// TIA Portal V17 export
// export: Created 2022-03-12T16:05:14.4802115Z, ExportSetting WithDefaults, DisplayName Totally Integrated Automation Portal, DisplayVersion V17, DisplayName TIA Portal Openness, DisplayVersion V17, DisplayName TIA Portal Version Control Interface, DisplayVersion V17, DisplayName STEP 7 Professional, DisplayVersion V17, DisplayName STEP 7 Safety, DisplayVersion V17, DisplayName WinCC Advanced / Unified PC, DisplayVersion V17
FUNCTION_BLOCK "UN_04_EventControl"   // FB31624, LAD
TITLE = UN_04_EventControl
{ S7_Optimized_Access := 'TRUE' }
AUTHOR : tech.team.motioncontrol@siemens.com
FAMILY : CPG
VERSION : 1.1
// Support: tech.team.motioncontrol@siemens.com
// stored: AutoNumber true, IsIECCheckEnabled false, IsRetainMemResEnabled false, MemoryReserve 100, SetENOAutomatically false, UDAEnableTagReadback false
   VAR
      instEventMgrAlarm { ExternalAccessible := 'False'; ExternalVisible := 'False'; ExternalWritable := 'False'; S7_SetPoint := 'True'} : "CPG_EventManager";   // instance FB - Event Manager - Alarms Events
      instEventMgrWarning { ExternalAccessible := 'False'; ExternalVisible := 'False'; ExternalWritable := 'False'; S7_SetPoint := 'True'} : "CPG_EventManager";   // instance FB - Event Manager - Warning Events
      instEventMgrStatus { ExternalAccessible := 'False'; ExternalVisible := 'False'; ExternalWritable := 'False'; S7_SetPoint := 'True'} : "CPG_EventManager";   // instance FB - Event Manager - Status Events
      instStatusAlarmsNotReset { ExternalAccessible := 'False'; ExternalVisible := 'False'; ExternalWritable := 'False'; S7_SetPoint := 'True'} : "CPG_Event";   // Status = Alarms Not Reset
      statEventMgr_Cmd_Reset { ExternalAccessible := 'False'; ExternalVisible := 'False'; ExternalWritable := 'False'} : Bool;   // Reset Cmd for event managers
      statEventMgr_Cmd_Clear1stFlt { ExternalAccessible := 'False'; ExternalVisible := 'False'; ExternalWritable := 'False'} : Bool;   // Clear 1st Fault Cmd for event managers
      statEventMgr_Clear1stFlt_OS { ExternalAccessible := 'False'; ExternalVisible := 'False'; ExternalWritable := 'False'} : Bool;   // Clear 1st Fault Cmd - One shot
   END_VAR
   VAR_TEMP   // added for the SCL form of the ladder/FBD networks
      _w1 : Bool;
      _w2 : Bool;
   END_VAR
BEGIN

REGION Network 2: ** STATE MODEL REPORTING STATUS ****
END_REGION

REGION Network 3: *** Call the PackML Module Initialize Logic ***
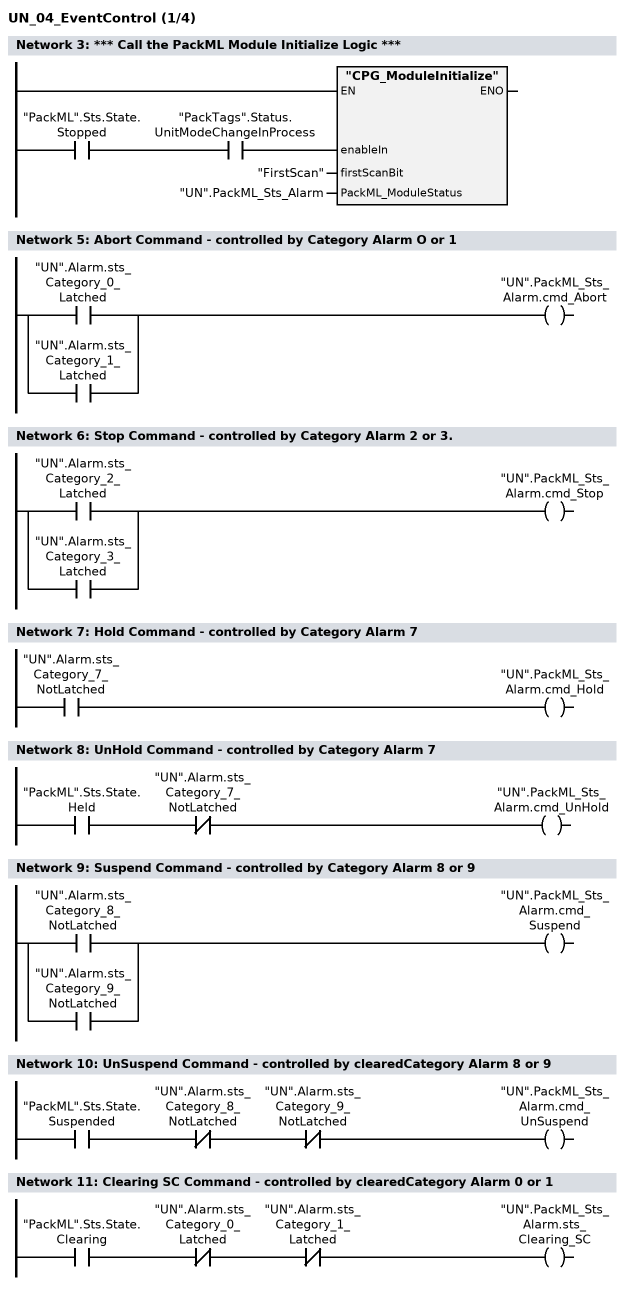
   RUNG wire#powerrail
      "CPG_ModuleInitialize"(enableIn := wire#w1, firstScanBit := "FirstScan", PackML_ModuleStatus := "UN".PackML_Sts_Alarm)
   END_RUNG
   RUNG wire#powerrail
      Contact( "PackML".Sts.State.Stopped )
      Contact( "PackTags".Status.UnitModeChangeInProcess )
   END_RUNG wire#w1
   // the same network as SCL:
   "CPG_ModuleInitialize"(enableIn := "PackML".Sts.State.Stopped AND "PackTags".Status.UnitModeChangeInProcess,
                          firstScanBit := "FirstScan",
                          PackML_ModuleStatus := "UN".PackML_Sts_Alarm);
END_REGION

REGION Network 4: Begin the LOGIC section.
END_REGION

REGION Network 5: Abort Command - controlled by Category Alarm O or 1
   RUNG wire#powerrail
      Contact( "UN".Alarm.sts_Category_0_Latched )
      wire#w1
      Coil( "UN".PackML_Sts_Alarm.cmd_Abort )
   END_RUNG
   RUNG wire#powerrail
      Contact( "UN".Alarm.sts_Category_1_Latched )
   END_RUNG wire#w1
   // the same network as SCL:
   "UN".PackML_Sts_Alarm.cmd_Abort := "UN".Alarm.sts_Category_0_Latched OR "UN".Alarm.sts_Category_1_Latched;
END_REGION

REGION Network 6: Stop Command - controlled by Category Alarm 2 or 3.
   RUNG wire#powerrail
      Contact( "UN".Alarm.sts_Category_2_Latched )
      wire#w1
      Coil( "UN".PackML_Sts_Alarm.cmd_Stop )
   END_RUNG
   RUNG wire#powerrail
      Contact( "UN".Alarm.sts_Category_3_Latched )
   END_RUNG wire#w1
   // the same network as SCL:
   "UN".PackML_Sts_Alarm.cmd_Stop := "UN".Alarm.sts_Category_2_Latched OR "UN".Alarm.sts_Category_3_Latched;
END_REGION

REGION Network 7: Hold Command - controlled by Category Alarm 7
   RUNG wire#powerrail
      Contact( "UN".Alarm.sts_Category_7_NotLatched )
      Coil( "UN".PackML_Sts_Alarm.cmd_Hold )
   END_RUNG
   // the same network as SCL:
   "UN".PackML_Sts_Alarm.cmd_Hold := "UN".Alarm.sts_Category_7_NotLatched;
END_REGION

REGION Network 8: UnHold Command - controlled by Category Alarm 7
   RUNG wire#powerrail
      Contact( "PackML".Sts.State.Held )
      I_Contact( "UN".Alarm.sts_Category_7_NotLatched )
      Coil( "UN".PackML_Sts_Alarm.cmd_UnHold )
   END_RUNG
   // the same network as SCL:
   "UN".PackML_Sts_Alarm.cmd_UnHold := "PackML".Sts.State.Held AND NOT "UN".Alarm.sts_Category_7_NotLatched;
END_REGION

REGION Network 9: Suspend Command - controlled by Category Alarm 8 or 9
   RUNG wire#powerrail
      Contact( "UN".Alarm.sts_Category_8_NotLatched )
      wire#w1
      Coil( "UN".PackML_Sts_Alarm.cmd_Suspend )
   END_RUNG
   RUNG wire#powerrail
      Contact( "UN".Alarm.sts_Category_9_NotLatched )
   END_RUNG wire#w1
   // the same network as SCL:
   "UN".PackML_Sts_Alarm.cmd_Suspend := "UN".Alarm.sts_Category_8_NotLatched OR "UN".Alarm.sts_Category_9_NotLatched;
END_REGION

REGION Network 10: UnSuspend Command - controlled by clearedCategory Alarm 8 or 9
   RUNG wire#powerrail
      Contact( "PackML".Sts.State.Suspended )
      I_Contact( "UN".Alarm.sts_Category_8_NotLatched )
      I_Contact( "UN".Alarm.sts_Category_9_NotLatched )
      Coil( "UN".PackML_Sts_Alarm.cmd_UnSuspend )
   END_RUNG
   // the same network as SCL:
   "UN".PackML_Sts_Alarm.cmd_UnSuspend := "PackML".Sts.State.Suspended AND NOT "UN".Alarm.sts_Category_8_NotLatched AND NOT "UN".Alarm.sts_Category_9_NotLatched;
END_REGION

REGION Network 11: Clearing SC Command - controlled by clearedCategory Alarm 0 or 1
   RUNG wire#powerrail
      Contact( "PackML".Sts.State.Clearing )
      I_Contact( "UN".Alarm.sts_Category_0_Latched )
      I_Contact( "UN".Alarm.sts_Category_1_Latched )
      Coil( "UN".PackML_Sts_Alarm.sts_Clearing_SC )
   END_RUNG
   // the same network as SCL:
   "UN".PackML_Sts_Alarm.sts_Clearing_SC := "PackML".Sts.State.Clearing AND NOT "UN".Alarm.sts_Category_0_Latched AND NOT "UN".Alarm.sts_Category_1_Latched;
END_REGION

REGION Network 12: Resetting S Command - controlled by clearedCategory Alarm 0-4
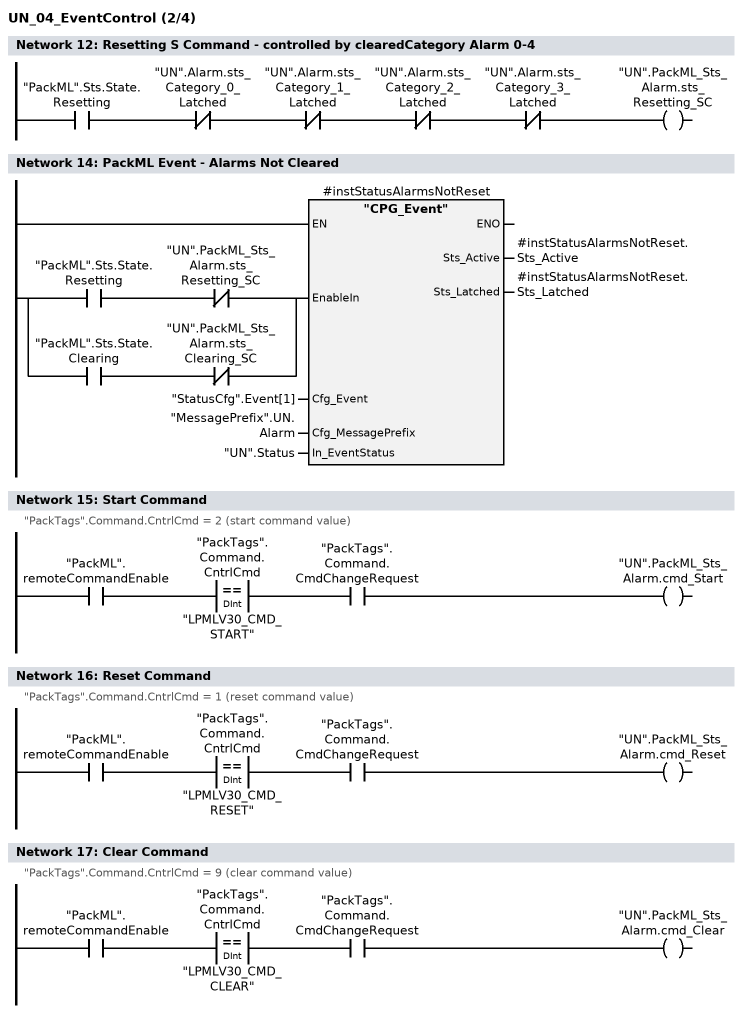
   RUNG wire#powerrail
      Contact( "PackML".Sts.State.Resetting )
      I_Contact( "UN".Alarm.sts_Category_0_Latched )
      I_Contact( "UN".Alarm.sts_Category_1_Latched )
      I_Contact( "UN".Alarm.sts_Category_2_Latched )
      I_Contact( "UN".Alarm.sts_Category_3_Latched )
      Coil( "UN".PackML_Sts_Alarm.sts_Resetting_SC )
   END_RUNG
   // the same network as SCL:
   "UN".PackML_Sts_Alarm.sts_Resetting_SC := "PackML".Sts.State.Resetting AND NOT "UN".Alarm.sts_Category_0_Latched AND NOT "UN".Alarm.sts_Category_1_Latched AND NOT "UN".Alarm.sts_Category_2_Latched AND NOT "UN".Alarm.sts_Category_3_Latched;
END_REGION

REGION Network 13: PackML Event -
END_REGION

REGION Network 14: PackML Event - Alarms Not Cleared
   RUNG wire#powerrail
      #instStatusAlarmsNotReset(EnableIn := wire#w1, Cfg_Event := "StatusCfg".Event[1], Cfg_MessagePrefix := "MessagePrefix".UN.Alarm, In_EventStatus := "UN".Status, Sts_Active => #instStatusAlarmsNotReset.Sts_Active, Sts_Latched => #instStatusAlarmsNotReset.Sts_Latched)
   END_RUNG
   RUNG wire#powerrail
      Contact( "PackML".Sts.State.Resetting )
      I_Contact( "UN".PackML_Sts_Alarm.sts_Resetting_SC )
   END_RUNG wire#w1
   RUNG wire#powerrail
      Contact( "PackML".Sts.State.Clearing )
      I_Contact( "UN".PackML_Sts_Alarm.sts_Clearing_SC )
   END_RUNG wire#w1
   // the same network as SCL:
   #instStatusAlarmsNotReset(EnableIn := ("PackML".Sts.State.Resetting AND NOT "UN".PackML_Sts_Alarm.sts_Resetting_SC) OR ("PackML".Sts.State.Clearing AND NOT "UN".PackML_Sts_Alarm.sts_Clearing_SC),   // "CPG_Event"
                           Cfg_Event := "StatusCfg".Event[1],
                           Cfg_MessagePrefix := "MessagePrefix".UN.Alarm,
                           In_EventStatus := "UN".Status,
                           Sts_Active => #instStatusAlarmsNotReset.Sts_Active,
                           Sts_Latched => #instStatusAlarmsNotReset.Sts_Latched);
END_REGION

REGION Network 15: Start Command
   // "PackTags".Command.CntrlCmd = 2 (start command value)
   RUNG wire#powerrail
      Contact( "PackML".remoteCommandEnable )
      { S7_Templates := "SrcType := DInt" } EQ_Contact(in1 := "PackTags".Command.CntrlCmd, in2 := "LPMLV30_CMD_START")
      Contact( "PackTags".Command.CmdChangeRequest )
      Coil( "UN".PackML_Sts_Alarm.cmd_Start )
   END_RUNG
   // the same network as SCL:
   "UN".PackML_Sts_Alarm.cmd_Start := "PackML".remoteCommandEnable AND ("PackTags".Command.CntrlCmd = "LPMLV30_CMD_START") AND "PackTags".Command.CmdChangeRequest;
END_REGION

REGION Network 16: Reset Command
   // "PackTags".Command.CntrlCmd = 1 (reset command value)
   RUNG wire#powerrail
      Contact( "PackML".remoteCommandEnable )
      { S7_Templates := "SrcType := DInt" } EQ_Contact(in1 := "PackTags".Command.CntrlCmd, in2 := "LPMLV30_CMD_RESET")
      Contact( "PackTags".Command.CmdChangeRequest )
      Coil( "UN".PackML_Sts_Alarm.cmd_Reset )
   END_RUNG
   // the same network as SCL:
   "UN".PackML_Sts_Alarm.cmd_Reset := "PackML".remoteCommandEnable AND ("PackTags".Command.CntrlCmd = "LPMLV30_CMD_RESET") AND "PackTags".Command.CmdChangeRequest;
END_REGION

REGION Network 17: Clear Command
   // "PackTags".Command.CntrlCmd = 9 (clear command value)
   RUNG wire#powerrail
      Contact( "PackML".remoteCommandEnable )
      { S7_Templates := "SrcType := DInt" } EQ_Contact(in1 := "PackTags".Command.CntrlCmd, in2 := "LPMLV30_CMD_CLEAR")
      Contact( "PackTags".Command.CmdChangeRequest )
      Coil( "UN".PackML_Sts_Alarm.cmd_Clear )
   END_RUNG
   // the same network as SCL:
   "UN".PackML_Sts_Alarm.cmd_Clear := "PackML".remoteCommandEnable AND ("PackTags".Command.CntrlCmd = "LPMLV30_CMD_CLEAR") AND "PackTags".Command.CmdChangeRequest;
END_REGION

REGION Network 18: *** EVENT CONTROL MANAGERS ***
END_REGION

REGION Network 19: Reset Command - for all event managers
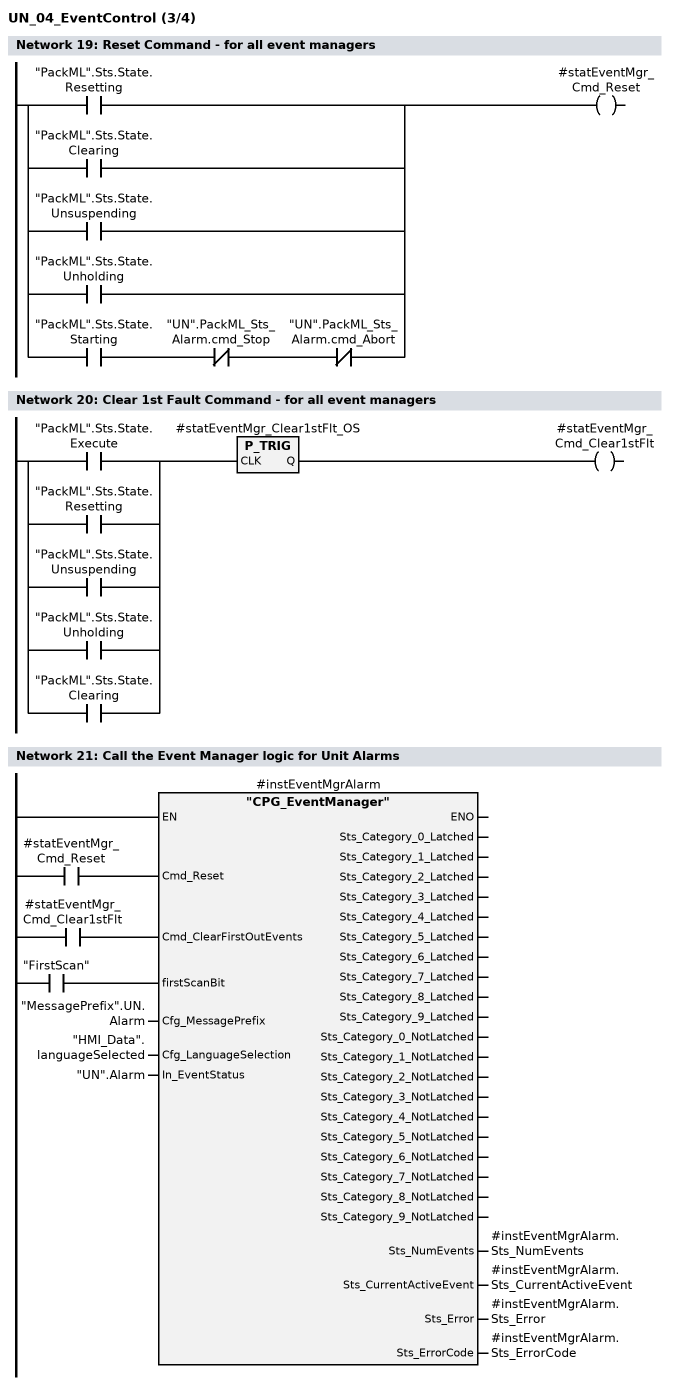
   RUNG wire#powerrail
      Contact( "PackML".Sts.State.Resetting )
      wire#w1
      Coil( #statEventMgr_Cmd_Reset )
   END_RUNG
   RUNG wire#powerrail
      Contact( "PackML".Sts.State.Clearing )
   END_RUNG wire#w1
   RUNG wire#powerrail
      Contact( "PackML".Sts.State.Unsuspending )
   END_RUNG wire#w1
   RUNG wire#powerrail
      Contact( "PackML".Sts.State.Unholding )
   END_RUNG wire#w1
   RUNG wire#powerrail
      Contact( "PackML".Sts.State.Starting )
      I_Contact( "UN".PackML_Sts_Alarm.cmd_Stop )
      I_Contact( "UN".PackML_Sts_Alarm.cmd_Abort )
   END_RUNG wire#w1
   // the same network as SCL:
   #statEventMgr_Cmd_Reset := "PackML".Sts.State.Resetting OR "PackML".Sts.State.Clearing OR "PackML".Sts.State.Unsuspending OR "PackML".Sts.State.Unholding OR ("PackML".Sts.State.Starting AND NOT "UN".PackML_Sts_Alarm.cmd_Stop AND NOT "UN".PackML_Sts_Alarm.cmd_Abort);
END_REGION

REGION Network 20: Clear 1st Fault Command - for all event managers
   RUNG wire#powerrail
      Contact( "PackML".Sts.State.Execute )
      wire#w1
      P_Trig( #statEventMgr_Clear1stFlt_OS )
      Coil( #statEventMgr_Cmd_Clear1stFlt )
   END_RUNG
   RUNG wire#powerrail
      Contact( "PackML".Sts.State.Resetting )
   END_RUNG wire#w1
   RUNG wire#powerrail
      Contact( "PackML".Sts.State.Unsuspending )
   END_RUNG wire#w1
   RUNG wire#powerrail
      Contact( "PackML".Sts.State.Unholding )
   END_RUNG wire#w1
   RUNG wire#powerrail
      Contact( "PackML".Sts.State.Clearing )
   END_RUNG wire#w1
   // the same network as SCL:
   #_w1 := "PackML".Sts.State.Execute OR "PackML".Sts.State.Resetting OR "PackML".Sts.State.Unsuspending OR "PackML".Sts.State.Unholding OR "PackML".Sts.State.Clearing;
   #_w2 := #_w1 AND NOT #statEventMgr_Clear1stFlt_OS;   // rising edge
   #statEventMgr_Clear1stFlt_OS := #_w1;
   #statEventMgr_Cmd_Clear1stFlt := #_w2;
END_REGION

REGION Network 21: Call the Event Manager logic for Unit Alarms
   RUNG wire#powerrail
      #instEventMgrAlarm(Cmd_Reset := wire#w1, Cmd_ClearFirstOutEvents := wire#w2, firstScanBit := wire#w3, Cfg_MessagePrefix := "MessagePrefix".UN.Alarm, Cfg_LanguageSelection := "HMI_Data".languageSelected, In_EventStatus := "UN".Alarm, Sts_Category_0_Latched =>, Sts_Category_1_Latched =>, Sts_Category_2_Latched =>, Sts_Category_3_Latched =>, Sts_Category_4_Latched =>, Sts_Category_5_Latched =>, Sts_Category_6_Latched =>, Sts_Category_7_Latched =>, Sts_Category_8_Latched =>, Sts_Category_9_Latched =>, Sts_Category_0_NotLatched =>, Sts_Category_1_NotLatched =>, Sts_Category_2_NotLatched =>, Sts_Category_3_NotLatched =>, Sts_Category_4_NotLatched =>, Sts_Category_5_NotLatched =>, Sts_Category_6_NotLatched =>, Sts_Category_7_NotLatched =>, Sts_Category_8_NotLatched =>, Sts_Category_9_NotLatched =>, Sts_NumEvents => #instEventMgrAlarm.Sts_NumEvents, Sts_CurrentActiveEvent => #instEventMgrAlarm.Sts_CurrentActiveEvent, Sts_Error => #instEventMgrAlarm.Sts_Error, Sts_ErrorCode => #instEventMgrAlarm.Sts_ErrorCode)
   END_RUNG
   RUNG wire#powerrail
      Contact( #statEventMgr_Cmd_Reset )
   END_RUNG wire#w1
   RUNG wire#powerrail
      Contact( #statEventMgr_Cmd_Clear1stFlt )
   END_RUNG wire#w2
   RUNG wire#powerrail
      Contact( "FirstScan" )
   END_RUNG wire#w3
   // the same network as SCL:
   #instEventMgrAlarm(Cmd_Reset := #statEventMgr_Cmd_Reset,   // "CPG_EventManager"
                      Cmd_ClearFirstOutEvents := #statEventMgr_Cmd_Clear1stFlt,
                      firstScanBit := "FirstScan",
                      Cfg_MessagePrefix := "MessagePrefix".UN.Alarm,
                      Cfg_LanguageSelection := "HMI_Data".languageSelected,
                      In_EventStatus := "UN".Alarm,
                      Sts_NumEvents => #instEventMgrAlarm.Sts_NumEvents,
                      Sts_CurrentActiveEvent => #instEventMgrAlarm.Sts_CurrentActiveEvent,
                      Sts_Error => #instEventMgrAlarm.Sts_Error,
                      Sts_ErrorCode => #instEventMgrAlarm.Sts_ErrorCode);
END_REGION

REGION Network 22: Call the Event Manager logic for Unit Warnings
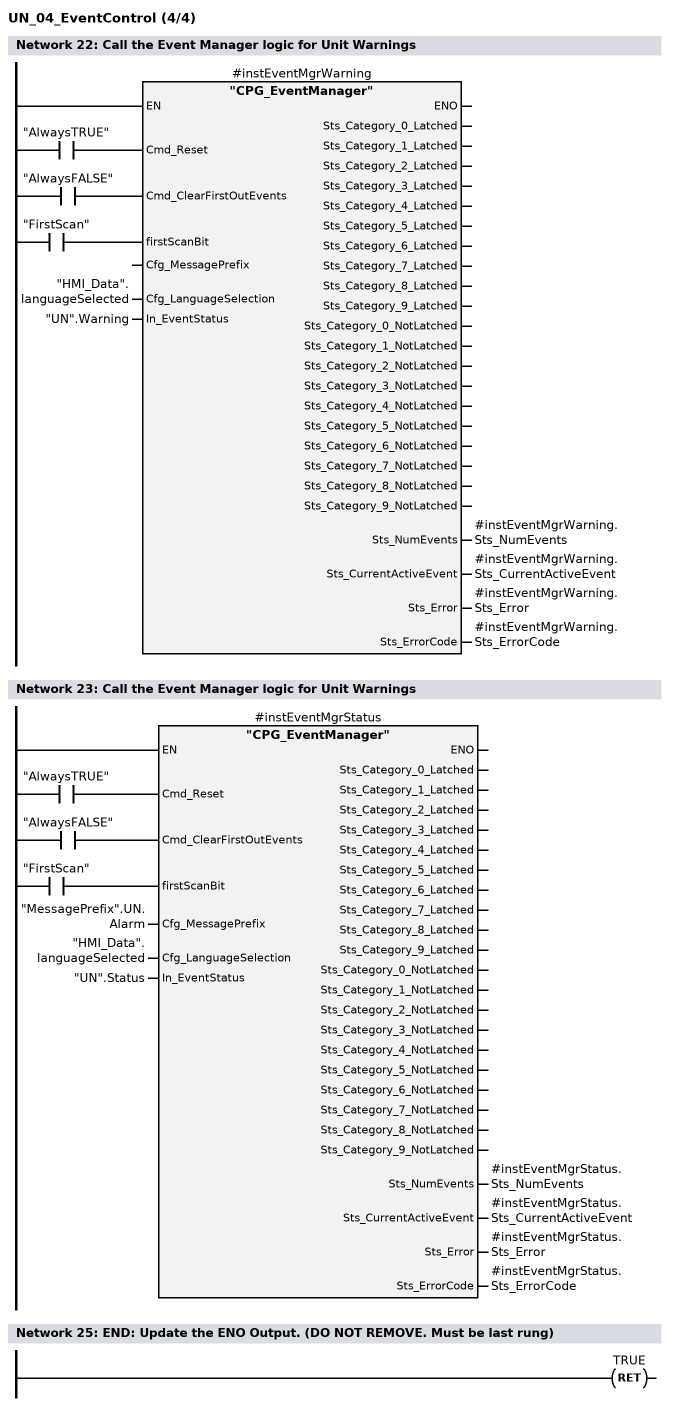
   RUNG wire#powerrail
      #instEventMgrWarning(Cmd_Reset := wire#w1, Cmd_ClearFirstOutEvents := wire#w2, firstScanBit := wire#w3, Cfg_MessagePrefix :=, Cfg_LanguageSelection := "HMI_Data".languageSelected, In_EventStatus := "UN".Warning, Sts_Category_0_Latched =>, Sts_Category_1_Latched =>, Sts_Category_2_Latched =>, Sts_Category_3_Latched =>, Sts_Category_4_Latched =>, Sts_Category_5_Latched =>, Sts_Category_6_Latched =>, Sts_Category_7_Latched =>, Sts_Category_8_Latched =>, Sts_Category_9_Latched =>, Sts_Category_0_NotLatched =>, Sts_Category_1_NotLatched =>, Sts_Category_2_NotLatched =>, Sts_Category_3_NotLatched =>, Sts_Category_4_NotLatched =>, Sts_Category_5_NotLatched =>, Sts_Category_6_NotLatched =>, Sts_Category_7_NotLatched =>, Sts_Category_8_NotLatched =>, Sts_Category_9_NotLatched =>, Sts_NumEvents => #instEventMgrWarning.Sts_NumEvents, Sts_CurrentActiveEvent => #instEventMgrWarning.Sts_CurrentActiveEvent, Sts_Error => #instEventMgrWarning.Sts_Error, Sts_ErrorCode => #instEventMgrWarning.Sts_ErrorCode)
   END_RUNG
   RUNG wire#powerrail
      Contact( "AlwaysTRUE" )
   END_RUNG wire#w1
   RUNG wire#powerrail
      Contact( "AlwaysFALSE" )
   END_RUNG wire#w2
   RUNG wire#powerrail
      Contact( "FirstScan" )
   END_RUNG wire#w3
   // the same network as SCL:
   #instEventMgrWarning(Cmd_Reset := "AlwaysTRUE",   // "CPG_EventManager"
                        Cmd_ClearFirstOutEvents := "AlwaysFALSE",
                        firstScanBit := "FirstScan",
                        Cfg_LanguageSelection := "HMI_Data".languageSelected,
                        In_EventStatus := "UN".Warning,
                        Sts_NumEvents => #instEventMgrWarning.Sts_NumEvents,
                        Sts_CurrentActiveEvent => #instEventMgrWarning.Sts_CurrentActiveEvent,
                        Sts_Error => #instEventMgrWarning.Sts_Error,
                        Sts_ErrorCode => #instEventMgrWarning.Sts_ErrorCode);
END_REGION

REGION Network 23: Call the Event Manager logic for Unit Warnings
   RUNG wire#powerrail
      #instEventMgrStatus(Cmd_Reset := wire#w1, Cmd_ClearFirstOutEvents := wire#w2, firstScanBit := wire#w3, Cfg_MessagePrefix := "MessagePrefix".UN.Alarm, Cfg_LanguageSelection := "HMI_Data".languageSelected, In_EventStatus := "UN".Status, Sts_Category_0_Latched =>, Sts_Category_1_Latched =>, Sts_Category_2_Latched =>, Sts_Category_3_Latched =>, Sts_Category_4_Latched =>, Sts_Category_5_Latched =>, Sts_Category_6_Latched =>, Sts_Category_7_Latched =>, Sts_Category_8_Latched =>, Sts_Category_9_Latched =>, Sts_Category_0_NotLatched =>, Sts_Category_1_NotLatched =>, Sts_Category_2_NotLatched =>, Sts_Category_3_NotLatched =>, Sts_Category_4_NotLatched =>, Sts_Category_5_NotLatched =>, Sts_Category_6_NotLatched =>, Sts_Category_7_NotLatched =>, Sts_Category_8_NotLatched =>, Sts_Category_9_NotLatched =>, Sts_NumEvents => #instEventMgrStatus.Sts_NumEvents, Sts_CurrentActiveEvent => #instEventMgrStatus.Sts_CurrentActiveEvent, Sts_Error => #instEventMgrStatus.Sts_Error, Sts_ErrorCode => #instEventMgrStatus.Sts_ErrorCode)
   END_RUNG
   RUNG wire#powerrail
      Contact( "AlwaysTRUE" )
   END_RUNG wire#w1
   RUNG wire#powerrail
      Contact( "AlwaysFALSE" )
   END_RUNG wire#w2
   RUNG wire#powerrail
      Contact( "FirstScan" )
   END_RUNG wire#w3
   // the same network as SCL:
   #instEventMgrStatus(Cmd_Reset := "AlwaysTRUE",   // "CPG_EventManager"
                       Cmd_ClearFirstOutEvents := "AlwaysFALSE",
                       firstScanBit := "FirstScan",
                       Cfg_MessagePrefix := "MessagePrefix".UN.Alarm,
                       Cfg_LanguageSelection := "HMI_Data".languageSelected,
                       In_EventStatus := "UN".Status,
                       Sts_NumEvents => #instEventMgrStatus.Sts_NumEvents,
                       Sts_CurrentActiveEvent => #instEventMgrStatus.Sts_CurrentActiveEvent,
                       Sts_Error => #instEventMgrStatus.Sts_Error,
                       Sts_ErrorCode => #instEventMgrStatus.Sts_ErrorCode);
END_REGION

REGION Network 25: END: Update the ENO Output. (DO NOT REMOVE. Must be last rung)
   RUNG wire#powerrail
      ReturnCoil( TRUE )
   END_RUNG
   // the same network as SCL:
   ENO := TRUE;
   RETURN;
END_REGION
END_FUNCTION_BLOCK
